// TIA Portal V17 export
// export: Created 2022-07-05T08:49:21.2209461Z, ExportSetting WithDefaults, DisplayName Totally Integrated Automation Portal, DisplayVersion V17, DisplayName TIA Portal Openness, DisplayVersion V17, DisplayName TIA Portal Version Control Interface, DisplayVersion V17, DisplayName STEP 7 Professional, DisplayVersion V17, DisplayName STEP 7 Safety, DisplayVersion V17, DisplayName WinCC Advanced, DisplayVersion V17
ORGANIZATION_BLOCK "Main"   // OB1, LAD, ProgramCycle
TITLE = "Main Program Sweep (Cycle)"
{ S7_Optimized_Access := 'TRUE' }
VERSION : 0.1
// stored: AutoNumber true, IsIECCheckEnabled false, SetENOAutomatically false
   VAR_INPUT
      Initial_Call : Bool;   // Initial call of this OB
      Remanence : Bool;   // =True, if remanent data are available
   END_VAR
BEGIN

REGION Network 1
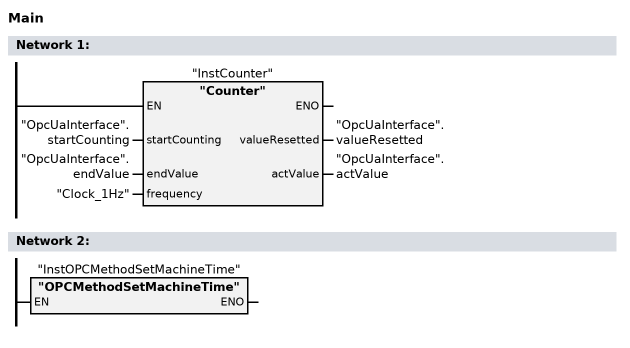
   RUNG wire#powerrail
      "InstCounter"(startCounting := "OpcUaInterface".startCounting, endValue := "OpcUaInterface".endValue, frequency := "Clock_1Hz", valueResetted => "OpcUaInterface".valueResetted, actValue => "OpcUaInterface".actValue)
   END_RUNG
   // the same network as SCL:
   "InstCounter"(startCounting := "OpcUaInterface".startCounting,   // "Counter"
                 endValue := "OpcUaInterface".endValue,
                 frequency := "Clock_1Hz",
                 valueResetted => "OpcUaInterface".valueResetted,
                 actValue => "OpcUaInterface".actValue);
END_REGION

REGION Network 2
   RUNG wire#powerrail
      "InstOPCMethodSetMachineTime"()
   END_RUNG
   // the same network as SCL:
   "InstOPCMethodSetMachineTime"();   // "OPCMethodSetMachineTime"
END_REGION
END_ORGANIZATION_BLOCK
